// TIA Portal V16 export
// export: Created 2021-04-06T19:52:12.4960301Z, ExportSetting WithDefaults, DisplayName Totally Integrated Automation Portal, DisplayVersion V16, DisplayName TIA Portal Version Control Interface, DisplayVersion V16, DisplayName TIA Portal Openness, DisplayVersion V16, DisplayName STEP 7 Professional, DisplayVersion V16, DisplayName STEP 7 Safety, DisplayVersion V16, DisplayName WinCC Unified SCADA Engineering System, DisplayVersion V16
FUNCTION "preIOtoDB" : Void   // FC3, LAD
{ S7_Optimized_Access := 'TRUE' }
VERSION : 0.1
// stored: AutoNumber true, IsIECCheckEnabled false, SetENOAutomatically false, UDAEnableTagReadback false
   VAR_TEMP
      i : Int;
      j : Int;
      k : Int;
      l : Int;
      "m" : Int;
   END_VAR
BEGIN

REGION Network 1 (SCL): активация катушек для автоматического и ручного режимов
   #i:=0;
   FOR #i := 1 TO 12 DO
       //Bunker_leftOpen
       IF "signalKVSStation".qManualMode.Bunker_leftOpen[#i] OR "signalKVSStation".qAutoMode.Bunker_leftOpen[#i]THEN
           "IO".output.Bunker_leftClose[#i] := true;
           "hmi".weightLine[#i].stateLeftValveWeightPocket := true;
       ELSE
           "IO".output.Bunker_leftClose[#i] := false;
       END_IF;

       //Bunker_leftClose
       IF "signalKVSStation".qManualMode.Bunker_leftClose[#i] OR "signalKVSStation".qAutoMode.Bunker_leftClose[#i] THEN
           "IO".output.Bunker_leftOpen[#i] := TRUE;
           "hmi".weightLine[#i].stateLeftValveWeightPocket := FALSE;
       ELSE
           "IO".output.Bunker_leftOpen[#i] := false;
       END_IF;

       //Bunker_rightOpen
       IF "signalKVSStation".qManualMode.Bunker_rightOpen[#i] OR "signalKVSStation".qAutoMode.Bunker_rightOpen[#i] THEN
           "IO".output.Bunker_rightClose[#i] := true;
           "hmi".weightLine[#i].stateRightValveWeightPocket := true;
       ELSE
           "IO".output.Bunker_rightClose[#i] := false;
       END_IF;

       //Bunker_rightClose
       IF "signalKVSStation".qManualMode.Bunker_rightClose[#i] OR "signalKVSStation".qAutoMode.Bunker_rightClose[#i] THEN
           "IO".output.Bunker_rightOpen[#i] := true;
           "hmi".weightLine[#i].stateRightValveWeightPocket := false;
       ELSE
           "IO".output.Bunker_rightOpen[#i] := false;
       END_IF;

       //Door_open
       IF "signalKVSStation".qManualMode.Door_open[#i] OR "signalKVSStation".qAutoMode.Door_open[#i] THEN
           "IO".output.Door_close[#i] := true;
           "hmi".weightLine[#i].stateValveAfterVibroLot := true;
       ELSE
           "IO".output.Door_close[#i] := false;
       END_IF;

       //Door_close
       IF "signalKVSStation".qManualMode.Door_close[#i] OR "signalKVSStation".qAutoMode.Door_close[#i] THEN
           "IO".output.Door_open[#i] := true;
           "hmi".weightLine[#i].stateValveAfterVibroLot := false;
       ELSE
           "IO".output.Door_open[#i] := false;
       END_IF;

       //vibroLot
       IF "signalKVSStation".qManualMode.vibroLot[#i] OR "signalKVSStation".qAutoMode.vibroLot[#i] THEN
           "IO".output.vibroLot[#i] := true;
           "hmi".weightLine[#i].isVibroLotWork := true;
       ELSE
           "hmi".weightLine[#i].isVibroLotWork := false;
           "IO".output.vibroLot[#i] := false;
       END_IF;

       //теперь все что на два цикла
       IF #i = 1 OR #i = 2 THEN
           //Yq_ReadyDoze
           IF "signalKVSStation".qManualMode.Yq_ReadyDoze[#i] OR "signalKVSStation".qAutoMode.Yq_ReadyDoze[#i] THEN
               "IO".output.Yq_ReadyDoze[#i] := true;
           ELSE
               "IO".output.Yq_ReadyDoze[#i] := false;
           END_IF;

           //Conv_FRV
           IF ("signalKVSStation".qManualMode.Conv_FRV[#i] OR "signalKVSStation".qAutoMode.Conv_FRV[#i]) AND NOT("IO".output.Conv_REV[#i])  THEN
               "IO".output.Conv_FRV[#i] := true;
           ELSE
               "IO".output.Conv_FRV[#i] := false;
           END_IF;

           //Conv_REV
           IF ("signalKVSStation".qManualMode.Conv_REV[#i] OR "signalKVSStation".qAutoMode.Conv_REV[#i]) AND NOT("IO".output.Conv_FRV[#i]) THEN
               "IO".output.Conv_REV[#i] := true;
           ELSE
               "IO".output.Conv_REV[#i] := false;
           END_IF;

           //Обратная связь по работе конвейера
           //
           IF "IO".output.Conv_FRV[#i] OR "IO".output.Conv_REV[#i] THEN
               "hmi".outConvAndPack[#i].isWorkConv := true;
           ELSE
               "hmi".outConvAndPack[#i].isWorkConv := false;
           END_IF;

           //vibroTable
           IF "signalKVSStation".qManualMode.vibroTable[#i] OR "signalKVSStation".qAutoMode.vibroTable[#i] THEN
               "IO".output.vibroTable[#i] := true;
               "hmi".addedVibro.stateVibroTable[#i] := true;
           ELSE
               "IO".output.vibroTable[#i] := false;
               "hmi".addedVibro.stateVibroTable[#i] := false;
           END_IF;


       END_IF;

       //flipper_Up
       IF "signalKVSStation".qManualMode.flipper_Up OR "signalKVSStation".qAutoMode.flipper_Up THEN
           "IO".output.flipper_Down := true;
           "hmi".plavnik.statePlavnik := true;
       ELSE
           "IO".output.flipper_Down := false;
       END_IF;

       //flipper_Down
       IF "signalKVSStation".qManualMode.flipper_Down OR "signalKVSStation".qAutoMode.flipper_Down THEN
           "IO".output.flipper_Up := true;
           "hmi".plavnik.statePlavnik := false;
       ELSE
           "IO".output.flipper_Up := false;
       END_IF;

       //питатель
       IF "signalKVSStation".qManualMode.startInConv OR "signalKVSStation".qAutoMode.startInConv THEN
           "IO".output.convSource := true;
           "hmi".sourceConv.isConvWork := true;
       ELSE
           "IO".output.convSource := false;
           "hmi".sourceConv.isConvWork := false;
       END_IF;

   END_FOR;
END_REGION
END_FUNCTION
